(* Schneider Machine Expert - Basic project Project1_Part3, file version 1.6.0.0 *)
(* ProjectInformations: Name=New project *)

HARDWARE
  Cpu 0: TM221M16R/G
  EthernetConfiguration: NetworkName=M221, IpAllocationMode=FixedAddress, IpAddress=0.0.0.0, SubnetMask=0.0.0.0
  SerialLineConfiguration: Baud=Baud19200, Parity=ParityEven, DataBits=DataBits8, StopBits=StopBits1, PhysicalMedium=PhysicalMediumRs485, TransmissionMode=TransmissionModeModbusRtu, SlaveId=1, Addressing=SlaveAddressing
  MastTask: UsePeriodScanMode=false, PeriodScan=100
  FastTask: Period=255
  CpuBehavior: StartingMode=StartAsPreviousState, AutoSaveRamOnEeprom=true, WatchdogPeriod=250

SYMBOLS  (address, symbol, comment, settings)
  %TM0        [Type=TP, Preset=5, Base=OneSecond]
  %C1         "Count down from 5"  [Preset=5]

POU Project1-Part1B
  (* SectionNumber=1 *)

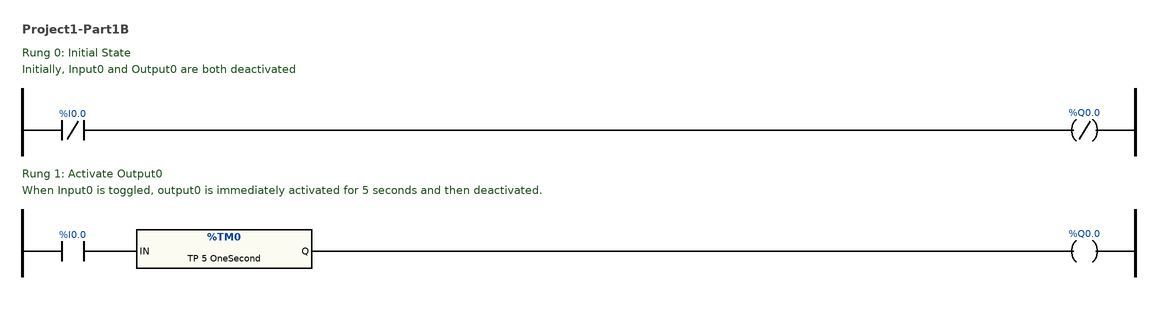

// Rung 0: Initial State
// Initially, Input0 and Output0 are both deactivated
  LDN %I0.0
  STN %Q0.0
  // as ST:
  //   %Q0.0 := NOT (NOT %I0.0);

// Rung 1: Activate Output0
// When Input0 is toggled, output0 is immediately activated for 5 seconds and then deactivated.
  BLK %TM0
  LD %I0.0
  IN
  OUT_BLK
  LD Q
  ST %Q0.0
  END_BLK
  // as ST:
  //   %TM0(IN := %I0.0);
  //   %Q0.0 := %TM0.Q;
